(* Schneider Machine Expert - Basic project buffer_station, file version 2.7.0.0 *)
(* ProjectInformations: Name=Nuevo proyecto *)

HARDWARE
  Cpu 0: TM221M16R/G
  EthernetConfiguration: NetworkName=M221, IpAllocationMode=FixedAddress, IpAddress=0.0.0.0, SubnetMask=0.0.0.0
  SerialLineConfiguration: Baud=Baud19200, Parity=ParityEven, DataBits=DataBits8, StopBits=StopBits1, PhysicalMedium=PhysicalMediumRs485, TransmissionMode=TransmissionModeModbusRtu, SlaveId=1, Addressing=SlaveAddressing
  MastTask: UsePeriodScanMode=false, PeriodScan=100
  FastTask: Period=255
  CpuBehavior: StartingMode=StartAsPreviousState, AutoSaveRamOnEeprom=true, WatchdogPeriod=250

SYMBOLS  (address, symbol, comment, settings)
  %M0         "At buffer entry"
  %M1         "At buffer exit"
  %M2         "At exit"
  %M3         "Start"
  %M4         "Reset"
  %M5         "Stop"
  %M6         "Auto"
  %M7         "Emergency Stop"
  %M8         "Running"
  %M9         "Stop blade"
  %M10        "Start light"
  %M11        "Reset light"
  %M12        "Stop light"
  %MW0        "Buffer Vel."
  %MW1        "Buffer conveyor"
  %MW2        "Exit conveyor"
  %MW3        "Counter"

POU Nuevo POU
  (* SectionNumber=1 *)

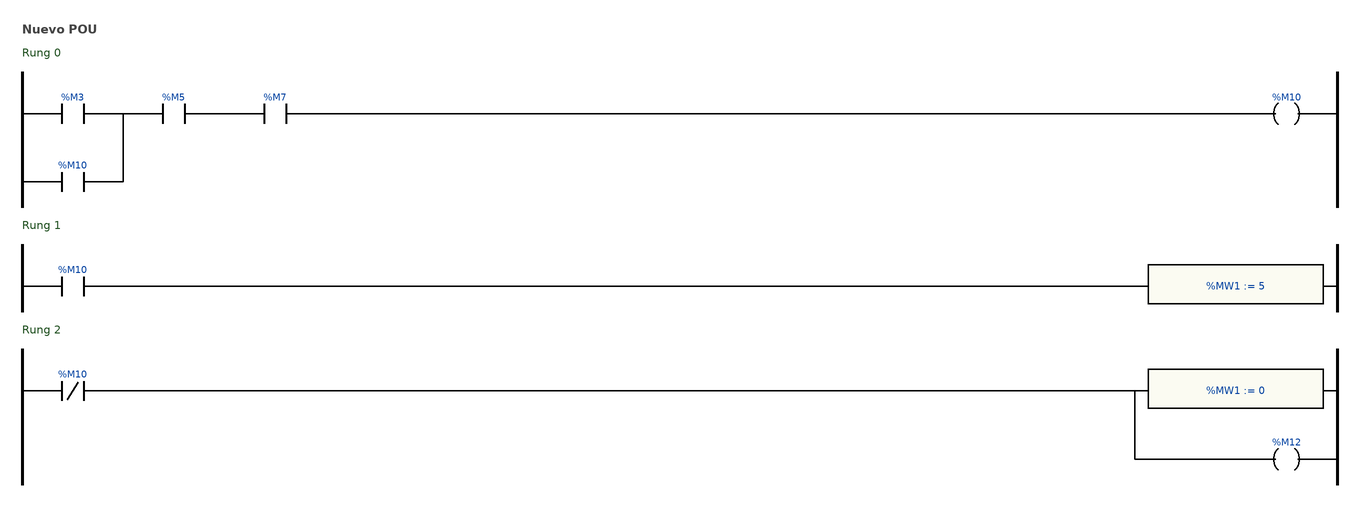

// Rung 0
  LD %M3
  OR %M10
  AND %M5
  AND %M7
  ST %M10
  // as ST:
  //   %M10 := (%M3 OR %M10) AND %M5 AND %M7;

// Rung 1
  LD %M10
  [ %MW1 := 5 ]
  // as ST:
  //   IF %M10 THEN %MW1 := 5; END_IF;

// Rung 2
  LDN %M10
  [ %MW1 := 0 ]
  ST %M12
  // as ST:
  //   IF NOT %M10 THEN %MW1 := 0; END_IF;
  //   %M12 := NOT %M10;
